(* Logix 5000 project; controller EuniceF_Lab1 vendor 1 type 14 code 150 rev 37.11; software revision 37.00 *)

TASK MainTask (continuous, watchdog 500 ms) : MainProgram

MODULES
   Local : vendor 1 type 14 code 150 (Compact 0, rev 37.11)
      Discrete_IO : Embedded (Compact 1, rev 3.1, Output RPI 20 ms)
      Analog_IO : Embedded (Compact 2, rev 1.1, Output RPI 80 ms)
      Counters : Embedded (Compact 3, rev 1.1, Output RPI 20 ms)
END_MODULES

VAR_GLOBAL   (* controller tags *)
   Countfor60cm : DINT;
   Default_Kfactor : DINT;
   Diif_Pressure : ALIAS FOR Local:2:O.Ch1Data;
   Done : ALIAS FOR Local:1:I.Data.15;
   DrainValve : ALIAS FOR Local:1:O.Data.10;
   Fill_Valve : ALIAS FOR Local:2:I.Ch1Data;
   Full : DINT;
   Full_Btn : ALIAS FOR Local:1:I.Data.13;
   Good : ALIAS FOR Local:1:I.Data.14;
   Half : DINT;
   Half_Btn : ALIAS FOR Local:1:I.Data.12;
   HSC1_CurentCount : ALIAS FOR Local:3:I.Ctr0CurrentCount;
   K_factor : DINT;
   LevelMax : DINT;
   LevelMin : DINT;
   Mixer : ALIAS FOR Local:1:O.Data.9;
   Prove : BOOL;
   Pump : ALIAS FOR Local:1:O.Data.8;
   Quarter : DINT;
   Quarter_Btn : ALIAS FOR Local:1:I.Data.11;
   Reset_HSC : ALIAS FOR Local:3:O.Ctr1SoftPreset;
   SEQ : DINT;
   Start : ALIAS FOR Local:1:I.Data.1;
   Status : STRING;
   Stop : ALIAS FOR Local:1:I.Data.2;
   T1 : TIMER := (PRE := 10000);
   Valve_Position : ALIAS FOR Local:2:O.Ch1Data;
END_VAR

PROGRAM MainProgram   (* main routine MainRoutine *)

ROUTINE MainRoutine   (* ladder *)
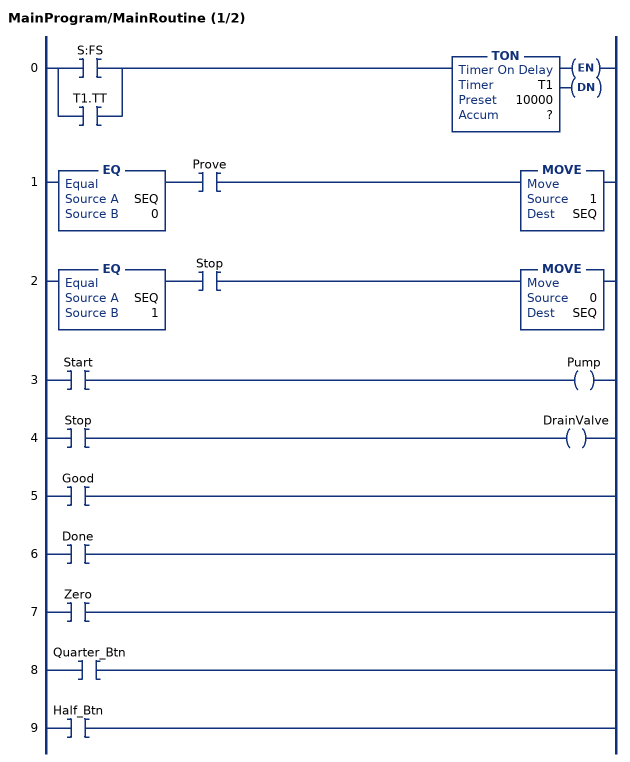
   0: [XIC(S:FS) ,XIC(T1.TT) ]TON(T1,?,?);
   1: EQ(SEQ,0)XIC(Prove)MOVE(1,SEQ);
   2: EQ(SEQ,1)XIC(Stop)MOVE(0,SEQ);
   3: XIC(Start)OTE(Pump);
   4: XIC(Stop)OTE(DrainValve);
   5: XIC(Good);
   6: XIC(Done);
   7: XIC(Zero);
   8: XIC(Quarter_Btn);
   9: XIC(Half_Btn);
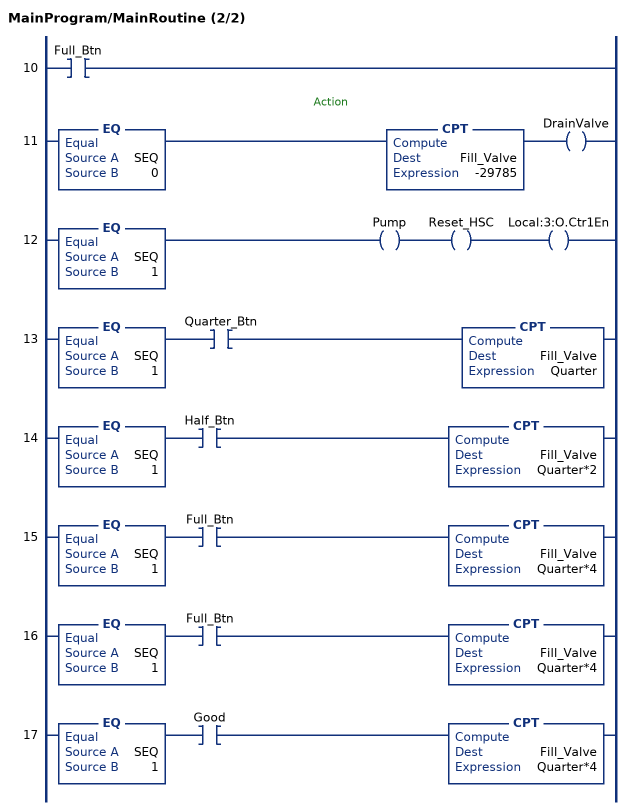
   10: XIC(Full_Btn);
   // Action
   11: EQ(SEQ,0)CPT(Fill_Valve,-29785)OTE(DrainValve);
   12: EQ(SEQ,1)OTE(Pump)OTE(Reset_HSC)OTE(Local:3:O.Ctr1En);
   13: EQ(SEQ,1)XIC(Quarter_Btn)CPT(Fill_Valve,Quarter);
   14: EQ(SEQ,1)XIC(Half_Btn)CPT(Fill_Valve,Quarter*2);
   15: EQ(SEQ,1)XIC(Full_Btn)CPT(Fill_Valve,Quarter*4);
   16: EQ(SEQ,1)XIC(Full_Btn)CPT(Fill_Valve,Quarter*4);
   17: EQ(SEQ,1)XIC(Good)CPT(Fill_Valve,Quarter*4);
END_ROUTINE
END_PROGRAM
